(* PLC project CoDeSys External Library Template, WAGO e!COCKPIT e!COCKPIT, author 3S - Smart Software Solutions GmbH *)
(* stored: creationDateTime 2019-10-29T12:37:19.9144384, version 3.5.5.30, modificationDateTime 2019-10-29T12:36:39.3744516, organization 3S - Smart Software Solutions GmbH *)
(* Library project template with all possible element types, docu and a sample project structure *)

FUNCTION fnKonwersja2x16naFloat32BySchneider : BOOL
  VAR_INPUT
    wRejestrMSW : WORD;  (* MSW - Most Significant Word *)
    wRejestrLSW : WORD;  (* LSW - Least Significant Word *)
  END_VAR
  VAR_IN_OUT
    rWartoscFloat32 : REAL;
  END_VAR
  VAR
    rZnak : REAL;
    rTempMSW : REAL;
    rTempMSW2 : REAL;
    wTempMSW : WORD;
    wTempMSW2 : WORD;
    dwTemp : DWORD;
    lrStala1 : LREAL := 8388608.0;
    lrStala2 : LREAL := 4194304.0;
    lrTemp : LREAL;
    rFaction : REAL;
    rExponent : REAL;
  END_VAR

            (*			
Autor:					Paweł Kąkol, 
Prawa majątkowe: 		Solwena Sp. z o.o., 
Aktualizacje:			2017-11-03-13:45-PK

Opis:					Funkcja do konwersji 2 rejestrów modbusowych na zmienną Float32 by Schneider Electric
*)
wTempMSW := wRejestrMSW / 256; // wyciagniecie 8 starszych bitow
//ustalanie znaku
IF (wTempMSW AND 128) = 128 THEN
	rZnak := -1.0;
	wTempMSW := wTempMSW AND 127; // usuniecie bitu znaku
ELSE
	rZnak := 1.0;
END_IF
wTempMSW2 := wRejestrMSW MOD 256; // wyciagniecie 8 mlodszych bitow
wTempMSW := (wTempMSW * 2) + ((wTempMSW2 AND 128) / 128); //przesuniecie bitowe o 1 w lewo wraz z dodaniem na najmlodsza pozycje najstarszego bitu z młodszych 8 bitow
wTempMSW2 := wTempMSW2 AND 127;// usuniecie najstarszego bitu
rExponent := WORD_TO_REAL(wTempMSW) - 127.0; // wyznaczanie wykladnika
dwTemp := WORD_TO_DWORD(wTempMSW2); //konwersja zmiennej 16-bitowej na 32-bitowa
dwTemp := dwTemp * 65536; //przesuniecie bitowe w lewo o 16 pozycji
dwTemp := dwTemp + WORD_TO_DWORD(wRejestrLSW); // dostawienie na koncu 16 bitow zmiennej LSW
lrTemp := DWORD_TO_LREAL(dwTemp);
//wybieranie ulamka
IF wTempMSW > 0 THEN
	rFaction := LREAL_TO_REAL((lrTemp / lrStala1) + 1.0);
ELSE
	rFaction := LREAL_TO_REAL(lrTemp / lrStala2);
END_IF
//obliczanie wartosci Float32
rWartoscFloat32 := rZnak * rFaction * EXPT(2.0, rExponent);
          
END_FUNCTION
